PROGRAM SaveDatabase
VAR
	fbPLCDBWrite : FB_PLCDBWriteEvt (sNetID := '', tTimeout := T#5S);
	myDBID : UDINT:=1;
	sMyTableName : T_MaxString:='Data';
	ColumnNames : ARRAY [0..91] OF STRING(50);
	insertData : aS_DBField;
	tcMessage : I_TcMessage;
	
	//Các biến tạo timestamp
	systime: GETSYSTEMTIME;
	currentTime: T_FILETIME;
	timestring: string;
	
	bFirstScan: BOOL;
	bExecute: BOOL;
	fbTon: TON;
	iID: LINT;
END_VAR

IF NOT bFirstScan THEN
	bFirstScan := TRUE;
	InitColumnNames();
END_IF

fbTon(IN:= NOT fbTon.Q, PT:= T#1S);	
IF fbTon.Q THEN
	UpdateData();
	bExecute := TRUE;
END_IF

IF bExecute AND bFirstScan THEN
	//UpdateData();
	IF fbPLCDBWrite.WriteStruct(
		hDBID:= myDBID,
		sTableName:= sMyTableName,
		pRecord:= ADR(insertData),
		cbRecord:= SIZEOF(insertData),
		pColumnNames:= ADR(ColumnNames) ,
		cbColumnNames:= SIZEOF(ColumnNames)
	)
	THEN
		IF fbPLCDBWrite.bError THEN
			tcMessage := fbPLCDBWrite.ipTcResult;
		ELSE
			iId := iId + 1;
			bExecute:= FALSE;
		END_IF
	END_IF	
	
END_IF

ACTION InitColumnNames:
ColumnNames[0] := 'Id';
ColumnNames[1] := 'Sync';
ColumnNames[2] := 'Timestamp';

ColumnNames[3] := 'FurTemp';
ColumnNames[4] := 'FurInper';
ColumnNames[5] := 'LphTemp';
ColumnNames[6] := 'LphPress';
ColumnNames[7] := 'LphInpress';
ColumnNames[8] := 'LphInflow';
ColumnNames[9] := 'DeaTemp';
ColumnNames[10] := 'DeaPress';
ColumnNames[11] := 'HphTemp';
ColumnNames[12] := 'HphPress';
ColumnNames[13] := 'HphInpress';
ColumnNames[14] := 'HphInflow';
ColumnNames[15] := 'BoiTemp';
ColumnNames[16] := 'BoiPress';
ColumnNames[17] := 'ConTemp';
ColumnNames[18] := 'ConInflow';
ColumnNames[19] := 'TurHtemp';
ColumnNames[20] := 'TurItemp';
ColumnNames[21] := 'TurLtemp';
ColumnNames[22] := 'TurHpress';
ColumnNames[23] := 'TurIpress';
ColumnNames[24] := 'TurLpress';
ColumnNames[25] := 'TurSpeed';

ColumnNames[26] := 'PconMode';
ColumnNames[27] := 'PconRun';
ColumnNames[28] := 'PconVal';
ColumnNames[29] := 'PconTime';
ColumnNames[30] := 'PconAtime';
ColumnNames[31] := 'PconFault';

ColumnNames[32] := 'PsupMode';
ColumnNames[33] := 'PsupRun';
ColumnNames[34] := 'PsupVal';
ColumnNames[35] := 'PsupTime';
ColumnNames[36] := 'PsupAtime';
ColumnNames[37] := 'PsupFault';

ColumnNames[38] := 'PcirMode';
ColumnNames[39] := 'PcirRun';
ColumnNames[40] := 'PcirVal';
ColumnNames[41] := 'PcirTime';
ColumnNames[42] := 'PcirAtime';
ColumnNames[43] := 'PcirFault';

ColumnNames[44] := 'F1Mode';
ColumnNames[45] := 'F1Run';
ColumnNames[46] := 'F1Val';
ColumnNames[47] := 'F1Time';
ColumnNames[48] := 'F1Atime';
ColumnNames[49] := 'F1Fault';

ColumnNames[50] := 'F2Mode';
ColumnNames[51] := 'F2Run';
ColumnNames[52] := 'F2Val';
ColumnNames[53] := 'F2Time';
ColumnNames[54] := 'F2Atime';
ColumnNames[55] := 'F2Fault';

ColumnNames[56] := 'F3Mode';
ColumnNames[57] := 'F3Run';
ColumnNames[58] := 'F3Val';
ColumnNames[59] := 'F3Time';
ColumnNames[60] := 'F3Atime';
ColumnNames[61] := 'F3Fault';

ColumnNames[62] := 'VlphMode';
ColumnNames[63] := 'VlphRun';
ColumnNames[64] := 'VlphVal';
ColumnNames[65] := 'VlphTime';
ColumnNames[66] := 'VlphAtime';
ColumnNames[67] := 'VlphFault';

ColumnNames[68] := 'VdeaMode';
ColumnNames[69] := 'VdeaRun';
ColumnNames[70] := 'VdeaVal';
ColumnNames[71] := 'VdeaTime';
ColumnNames[72] := 'VdeaAtime';
ColumnNames[73] := 'VdeaFault';

ColumnNames[74] := 'VhphMode';
ColumnNames[75] := 'VhphRun';
ColumnNames[76] := 'VhphVal';
ColumnNames[77] := 'VhphTime';
ColumnNames[78] := 'VhphAtime';
ColumnNames[79] := 'VhphFault';

ColumnNames[80] := 'VturMode';
ColumnNames[81] := 'VturRun';
ColumnNames[82] := 'VturVal';
ColumnNames[83] := 'VturTime';
ColumnNames[84] := 'VturAtime';
ColumnNames[85] := 'VturFault';

ColumnNames[86] := 'PintMode';
ColumnNames[87] := 'PintRun';
ColumnNames[88] := 'PintVal';
ColumnNames[89] := 'PintTime';
ColumnNames[90] := 'PintAtime';
ColumnNames[91] := 'PintFault';
END_ACTION

ACTION UpdateData:
systime(timeLoDW => currentTime.dwLowDateTime, timeHiDW => currentTime.dwHighDateTime);	
timestring:= DT_TO_STRING(FILETIME_TO_DT(currentTime));
timestring:= delete(timestring, 3, 1);
timestring:= replace(timestring, ' ', 1, 11);

insertData.Id := iID;
insertData.Sync := FALSE;
insertData.Timestamp:= FILETIME_TO_DT(currentTime);
insertData.FurTemp:= Interfacex.ScadaInterface.Components.Furnace.Temperature;
insertData.FurInper:= Interfacex.ScadaInterface.Components.Furnace.InPercent;
insertData.LphTemp:= Interfacex.ScadaInterface.Components.LPHeater.Temperature;
insertData.LphPress:= Interfacex.ScadaInterface.Components.LPHeater.Pressure;
insertData.LphInpress:= Interfacex.ScadaInterface.Components.LPHeater.InPressure;
insertData.LphInflow:= Interfacex.ScadaInterface.Components.LPHeater.InFlow;
insertData.DeaTemp:= Interfacex.ScadaInterface.Components.Deaerator.Temperature;
insertData.DeaPress:= Interfacex.ScadaInterface.Components.Deaerator.Pressure;
insertData.HphTemp:= Interfacex.ScadaInterface.Components.HPHeater.Temperature;
insertData.HphPress:= Interfacex.ScadaInterface.Components.HPHeater.Pressure;
insertData.HphInpress:= Interfacex.ScadaInterface.Components.HPHeater.InPressure;
insertData.HphInflow:= Interfacex.ScadaInterface.Components.HPHeater.InFlow;
insertData.BoiTemp:= Interfacex.ScadaInterface.Components.Boiler.Temperature;
insertData.BoiPress:= Interfacex.ScadaInterface.Components.Boiler.Pressure;
insertData.ConTemp:= Interfacex.ScadaInterface.Components.Condenser.Temperature;
insertData.ConInflow:= Interfacex.ScadaInterface.Components.Condenser.InFlow;
insertData.TurHtemp:= Interfacex.ScadaInterface.Components.Turbine.HighTemperature;
insertData.TurItemp:= Interfacex.ScadaInterface.Components.Turbine.ImmediateTemperature;
insertData.TurLtemp:= Interfacex.ScadaInterface.Components.Turbine.OutTemperature;
insertData.TurHpress:= Interfacex.ScadaInterface.Components.Turbine.HighPressure;
insertData.TurIpress:= Interfacex.ScadaInterface.Components.Turbine.ImmediatePressure;
insertData.TurLpress:= Interfacex.ScadaInterface.Components.Turbine.OutPressure;
insertData.TurSpeed:= Interfacex.ScadaInterface.Components.Turbine.Rotation;

insertData.PconMode:= INT_TO_BYTE(Interfacex.ScadaInterface.Components.CondensePump.Mode); 
insertData.PconRun:= Interfacex.ScadaInterface.Components.CondensePump.RunFeedback;
insertData.PconVal:= Interfacex.ScadaInterface.Components.CondensePump.ActualSpeed;
insertData.PconTime:= Interfacex.ScadaInterface.Components.CondensePump.Runtime;
insertData.PconAtime:= Interfacex.ScadaInterface.Components.CondensePump.AccRuntime;
insertData.PconFault:= Interfacex.ScadaInterface.Components.CondensePump.Fault;

insertData.PsupMode:= INT_TO_BYTE(Interfacex.ScadaInterface.Components.SupplyPump.Mode); 
insertData.PsupRun:= Interfacex.ScadaInterface.Components.SupplyPump.RunFeedback;
insertData.PsupVal:= Interfacex.ScadaInterface.Components.SupplyPump.ActualSpeed;
insertData.PsupTime:= Interfacex.ScadaInterface.Components.SupplyPump.Runtime;
insertData.PsupAtime:= Interfacex.ScadaInterface.Components.SupplyPump.AccRuntime;
insertData.PsupFault:= Interfacex.ScadaInterface.Components.SupplyPump.Fault;

insertData.PcirMode:= INT_TO_BYTE(Interfacex.ScadaInterface.Components.CircularPump.Mode); 
insertData.PcirRun:= Interfacex.ScadaInterface.Components.CircularPump.RunFeedback;
insertData.PcirVal:= Interfacex.ScadaInterface.Components.CircularPump.ActualSpeed;
insertData.PcirTime:= Interfacex.ScadaInterface.Components.CircularPump.Runtime;
insertData.PcirAtime:= Interfacex.ScadaInterface.Components.CircularPump.AccRuntime;
insertData.PcirFault:= Interfacex.ScadaInterface.Components.CircularPump.Fault;

insertData.F1Mode:= INT_TO_BYTE(Interfacex.ScadaInterface.Components.ForceFan1.Mode); 
insertData.F1Run:= Interfacex.ScadaInterface.Components.ForceFan1.RunFeedback;
insertData.F1Val:= Interfacex.ScadaInterface.Components.ForceFan1.ActualSpeed;
insertData.F1Time:= Interfacex.ScadaInterface.Components.ForceFan1.Runtime;
insertData.F1Atime:= Interfacex.ScadaInterface.Components.ForceFan1.AccRuntime;
insertData.F1Fault:= Interfacex.ScadaInterface.Components.ForceFan1.Fault;

insertData.F2Mode:= INT_TO_BYTE(Interfacex.ScadaInterface.Components.ForceFan2.Mode); 
insertData.F2Run:= Interfacex.ScadaInterface.Components.ForceFan2.RunFeedback;
insertData.F2Val:= Interfacex.ScadaInterface.Components.ForceFan2.ActualSpeed;
insertData.F2Time:= Interfacex.ScadaInterface.Components.ForceFan2.Runtime;
insertData.F2Atime:= Interfacex.ScadaInterface.Components.ForceFan2.AccRuntime;
insertData.F2Fault:= Interfacex.ScadaInterface.Components.ForceFan2.Fault;

insertData.F3Mode:= INT_TO_BYTE(Interfacex.ScadaInterface.Components.ForceFan3.Mode); 
insertData.F3Run:= Interfacex.ScadaInterface.Components.ForceFan3.RunFeedback;
insertData.F3Val:= Interfacex.ScadaInterface.Components.ForceFan3.ActualSpeed;
insertData.F3Time:= Interfacex.ScadaInterface.Components.ForceFan3.Runtime;
insertData.F3Atime:= Interfacex.ScadaInterface.Components.ForceFan3.AccRuntime;
insertData.F3Fault:= Interfacex.ScadaInterface.Components.ForceFan3.Fault;

insertData.VlphMode:= INT_TO_BYTE(Interfacex.ScadaInterface.Components.LPHValve.Mode); 
insertData.VlphRun:= Interfacex.ScadaInterface.Components.LPHValve.RunFeedback;
insertData.VlphVal:= Interfacex.ScadaInterface.Components.LPHValve.OpenPercent;
insertData.VlphTime:= Interfacex.ScadaInterface.Components.LPHValve.Runtime;
insertData.VlphAtime:= Interfacex.ScadaInterface.Components.LPHValve.AccRuntime;
insertData.VlphFault:= Interfacex.ScadaInterface.Components.LPHValve.Fault;

insertData.VdeaMode:= INT_TO_BYTE(Interfacex.ScadaInterface.Components.AirEjValve.Mode); 
insertData.VdeaRun:= Interfacex.ScadaInterface.Components.AirEjValve.RunFeedback;
insertData.VdeaVal:= Interfacex.ScadaInterface.Components.AirEjValve.OpenPercent;
insertData.VdeaTime:= Interfacex.ScadaInterface.Components.AirEjValve.Runtime;
insertData.VdeaAtime:= Interfacex.ScadaInterface.Components.AirEjValve.AccRuntime;
insertData.VdeaFault:= Interfacex.ScadaInterface.Components.AirEjValve.Fault;

insertData.VhphMode:= INT_TO_BYTE(Interfacex.ScadaInterface.Components.HPHValve.Mode); 
insertData.VhphRun:= Interfacex.ScadaInterface.Components.HPHValve.RunFeedback;
insertData.VhphVal:= Interfacex.ScadaInterface.Components.HPHValve.OpenPercent;
insertData.VhphTime:= Interfacex.ScadaInterface.Components.HPHValve.Runtime;
insertData.VhphAtime:= Interfacex.ScadaInterface.Components.HPHValve.AccRuntime;
insertData.VhphFault:= Interfacex.ScadaInterface.Components.HPHValve.Fault;

insertData.VturMode:= INT_TO_BYTE(Interfacex.ScadaInterface.Components.TurbineValve.Mode); 
insertData.VturRun:= Interfacex.ScadaInterface.Components.TurbineValve.RunFeedback;
insertData.VturVal:= Interfacex.ScadaInterface.Components.TurbineValve.OpenPercent;
insertData.VturTime:= Interfacex.ScadaInterface.Components.TurbineValve.Runtime;
insertData.VturAtime:= Interfacex.ScadaInterface.Components.TurbineValve.AccRuntime;
insertData.VturFault:= Interfacex.ScadaInterface.Components.TurbineValve.Fault;

insertData.PintMode:= INT_TO_BYTE(Interfacex.ScadaInterface.Components.InterPump.Mode); 
insertData.PintRun:= Interfacex.ScadaInterface.Components.InterPump.RunFeedback;
insertData.PintVal:= Interfacex.ScadaInterface.Components.InterPump.ActualSpeed;
insertData.PintTime:= Interfacex.ScadaInterface.Components.InterPump.Runtime;
insertData.PintAtime:= Interfacex.ScadaInterface.Components.InterPump.AccRuntime;
insertData.PintFault:= Interfacex.ScadaInterface.Components.InterPump.Fault;
END_ACTION

END_PROGRAM

(* stored: Version 1.1.0.1, ProductVersion 3.1.4024.4
   POU SaveDatabase: Id {06944aa8-c996-4e22-9874-5e83ff9218ca}, SpecialFunc None
   Action InitColumnNames: Id {ca3a8eb2-aaef-4de3-a6b7-45fc2a26e24a}
   Action UpdateData: Id {ee102ece-0353-4bcb-bb58-75f20df150bc} *)
